FUNCTION_BLOCK PUBL_TEST (* Test PUBL_x in a Composite Function Block *)
  (* Standard: 61499-2 *)
  (* Version 0.0, 2002-12-17, JHC, Rockwell Automation *)
  (* Compiler header: package fb.rt.test; import fb.rt.net.*; *)
  (* Compiler Java IBM Jikes 1.06 *)
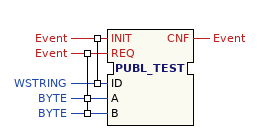
  EVENT_INPUT
    INIT WITH ID;
    REQ WITH A, B; (* Normal Execution Request *)
  END_EVENT
  EVENT_OUTPUT
    CNF; (* Execution Confirmation *)
  END_EVENT
  VAR_INPUT
    ID : WSTRING;
    A : BYTE;
    B : BYTE;
  END_VAR
  FBS
    TEST : PUBL_2;
  END_FBS
  EVENT_CONNECTIONS
    INIT TO TEST.INIT;
    REQ TO TEST.REQ;
    TEST.CNF TO CNF;
  END_CONNECTIONS
  DATA_CONNECTIONS
    ID TO TEST.ID;
    A TO TEST.SD_1;
    B TO TEST.SD_2;
  END_CONNECTIONS
END_FUNCTION_BLOCK
